_CFC_ (* Continuous Function Chart, elements in execution order *)
#0 INT_TO_REAL(SHU6_P2_TE1_AI1)
#1 DIV(#0, 10)
#2 SHU6_P2_TE1_VN <= #1
#3 I_GT_TE:ISTOK_GT(dost: TRUE, x: #1, ust: SHU6_P2_TE_HIGHLIMIT, shkal: -, gist: 1)
#4 I_LT_TE:ISTOK_LT(dost: TRUE, x: #1, ust: SHU6_P2_TE_LOWLIMIT, shkal: -, gist: 1)
#5 OR(#3.Xb, #4.Xm)
#6 TON_DOST:TON(IN: NOT #5, PT: T#10s)
#7 SHU6_P2_TE1_DOST <= #6.Q
#8 SUB(SHU6_P2_UST_SEZ_LETO, SHU6_P2_UST_SEZ_ZIMA)
#9 fb_SHU6_P2_TE1_B_UST_SEZ_LETO:ISTOK_GT(dost: #6.Q, x: #1, ust: SHU6_P2_UST_SEZ_LETO, shkal: -, gist: #8)
#10 SHU6_P2_TE1_B_UST_SEZ_LETO <= #9.Xb
#11 SHU6_P2_TE1_M_UST_SEZ_LETO <= #9.XbN
#12 fb_SHU6_P2_TE1_B_UST_MYAG_REG:ISTOK_GT(dost: #6.Q, x: #1, ust: SHU6_P2_UST_MYAG_REG, shkal: -, gist: 1)
#13 SHU6_P2_TE1_B_UST_MYAG_REG <= #12.Xb
#14 SHU6_P2_TE1_M_UST_MYAG_REG <= #12.XbN
_END_CFC_
(* the same logic as Structured Text *)
_t75 := INT_TO_REAL(SHU6_P2_TE1_AI1) / 10;
SHU6_P2_TE1_VN := _t75;
I_GT_TE(dost := TRUE, x := _t75, ust := SHU6_P2_TE_HIGHLIMIT, gist := 1);
I_LT_TE(dost := TRUE, x := _t75, ust := SHU6_P2_TE_LOWLIMIT, gist := 1);
TON_DOST(IN := NOT (I_GT_TE.Xb OR I_LT_TE.Xm), PT := T#10s);
SHU6_P2_TE1_DOST := TON_DOST.Q;
fb_SHU6_P2_TE1_B_UST_SEZ_LETO(dost := TON_DOST.Q, x := _t75, ust := SHU6_P2_UST_SEZ_LETO, gist := SHU6_P2_UST_SEZ_LETO - SHU6_P2_UST_SEZ_ZIMA);
SHU6_P2_TE1_B_UST_SEZ_LETO := fb_SHU6_P2_TE1_B_UST_SEZ_LETO.Xb;
SHU6_P2_TE1_M_UST_SEZ_LETO := fb_SHU6_P2_TE1_B_UST_SEZ_LETO.XbN;
fb_SHU6_P2_TE1_B_UST_MYAG_REG(dost := TON_DOST.Q, x := _t75, ust := SHU6_P2_UST_MYAG_REG, gist := 1);
SHU6_P2_TE1_B_UST_MYAG_REG := fb_SHU6_P2_TE1_B_UST_MYAG_REG.Xb;
SHU6_P2_TE1_M_UST_MYAG_REG := fb_SHU6_P2_TE1_B_UST_MYAG_REG.XbN;
END_PROGRAM

(* POU Input/AI/TE4, CFC *)
PROGRAM TE4
VAR
	TE4_YST: REAL;
	fb_TE4: ISTOK_ANALOGVH;
	ofset: REAL;
	fb_SHU6_P2_TE4_M_ZASCH: ISTOK_LT;
	fb_SHU6_P2_TE4_M_UST: ISTOK_LT;
	I_GT_TE: ISTOK_GT;
	I_LT_TE: ISTOK_LT;
	TON_DOST: TON;
END_VAR
VAR (* helpers for the ST form of the networks *)
	_t112 : REAL;
END_VAR
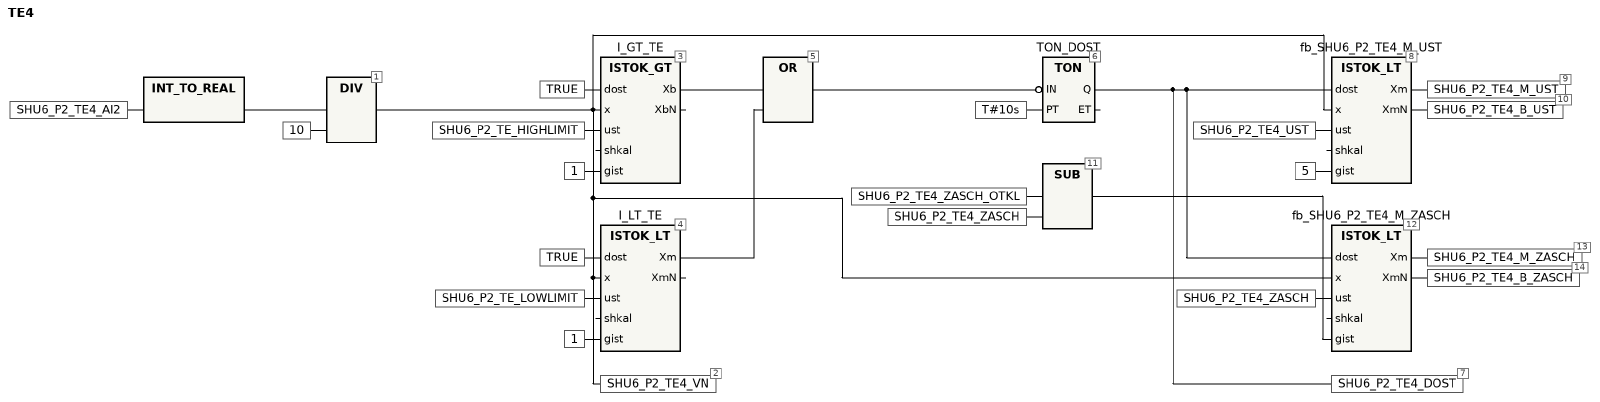
_CFC_ (* Continuous Function Chart, elements in execution order *)
#0 INT_TO_REAL(SHU6_P2_TE4_AI2)
#1 DIV(#0, 10)
#2 SHU6_P2_TE4_VN <= #1
#3 I_GT_TE:ISTOK_GT(dost: TRUE, x: #1, ust: SHU6_P2_TE_HIGHLIMIT, shkal: -, gist: 1)
#4 I_LT_TE:ISTOK_LT(dost: TRUE, x: #1, ust: SHU6_P2_TE_LOWLIMIT, shkal: -, gist: 1)
#5 OR(#3.Xb, #4.Xm)
#6 TON_DOST:TON(IN: NOT #5, PT: T#10s)
#7 SHU6_P2_TE4_DOST <= #6.Q
#8 fb_SHU6_P2_TE4_M_UST:ISTOK_LT(dost: #6.Q, x: #1, ust: SHU6_P2_TE4_UST, shkal: -, gist: 5)
#9 SHU6_P2_TE4_M_UST <= #8.Xm
#10 SHU6_P2_TE4_B_UST <= #8.XmN
#11 SUB(SHU6_P2_TE4_ZASCH_OTKL, SHU6_P2_TE4_ZASCH)
#12 fb_SHU6_P2_TE4_M_ZASCH:ISTOK_LT(dost: #6.Q, x: #1, ust: SHU6_P2_TE4_ZASCH, shkal: -, gist: #11)
#13 SHU6_P2_TE4_M_ZASCH <= #12.Xm
#14 SHU6_P2_TE4_B_ZASCH <= #12.XmN
_END_CFC_
(* the same logic as Structured Text *)
_t112 := INT_TO_REAL(SHU6_P2_TE4_AI2) / 10;
SHU6_P2_TE4_VN := _t112;
I_GT_TE(dost := TRUE, x := _t112, ust := SHU6_P2_TE_HIGHLIMIT, gist := 1);
I_LT_TE(dost := TRUE, x := _t112, ust := SHU6_P2_TE_LOWLIMIT, gist := 1);
TON_DOST(IN := NOT (I_GT_TE.Xb OR I_LT_TE.Xm), PT := T#10s);
SHU6_P2_TE4_DOST := TON_DOST.Q;
fb_SHU6_P2_TE4_M_UST(dost := TON_DOST.Q, x := _t112, ust := SHU6_P2_TE4_UST, gist := 5);
SHU6_P2_TE4_M_UST := fb_SHU6_P2_TE4_M_UST.Xm;
SHU6_P2_TE4_B_UST := fb_SHU6_P2_TE4_M_UST.XmN;
fb_SHU6_P2_TE4_M_ZASCH(dost := TON_DOST.Q, x := _t112, ust := SHU6_P2_TE4_ZASCH, gist := SHU6_P2_TE4_ZASCH_OTKL - SHU6_P2_TE4_ZASCH);
SHU6_P2_TE4_M_ZASCH := fb_SHU6_P2_TE4_M_ZASCH.Xm;
SHU6_P2_TE4_B_ZASCH := fb_SHU6_P2_TE4_M_ZASCH.XmN;
END_PROGRAM

(* POU Input/CI/MV2_1_OB, CFC *)
PROGRAM MV2_1_OB
VAR
	fb_M1_OBRbSM: ISTOK_GT;
	fb_M1b30: ISTOK_GT;
	fb_M1_OBRb45: ISTOK_GT;
	fb_M1_OBRm0_1: ISTOK_LT;
	fb_M_OBR: ISTOK_ANALOGVH;
	ofset: INT := 0;
	SR_DOST_M1: RS;
	dost_ton: TON;
END_VAR
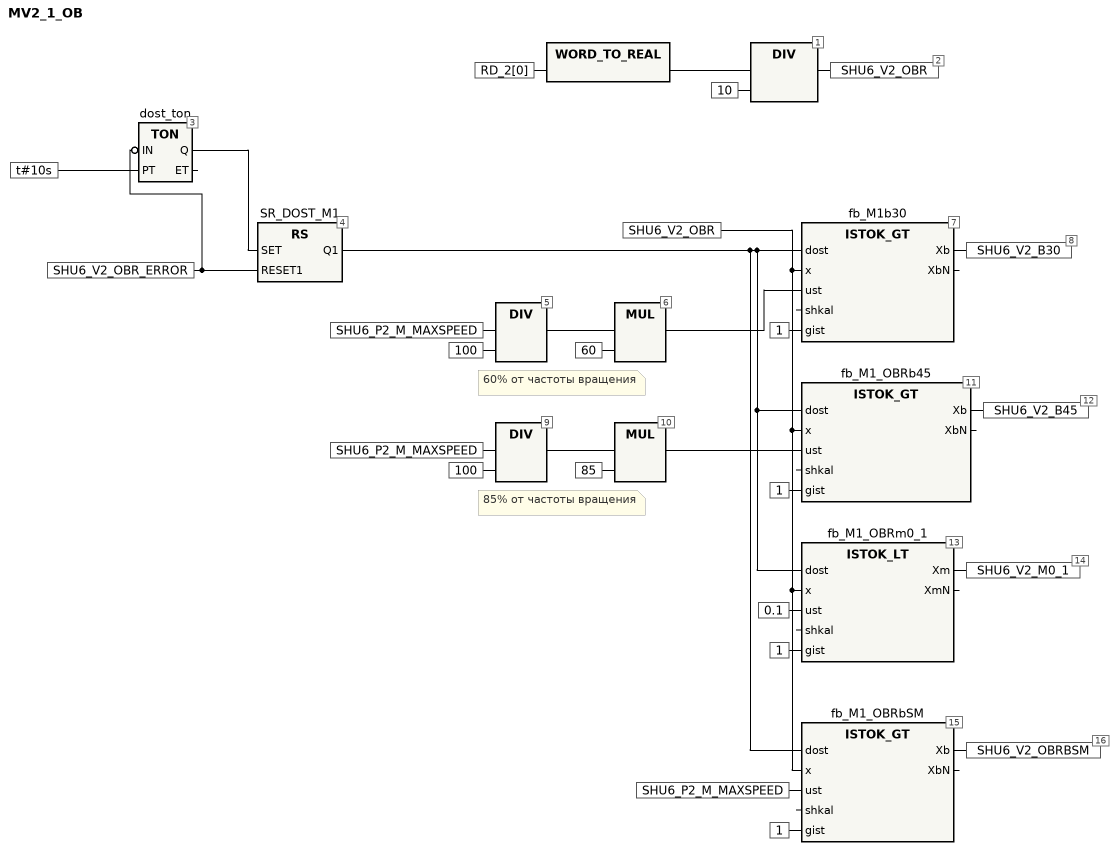
_CFC_ (* Continuous Function Chart, elements in execution order *)
(* 85% от частоты вращения *)
(* 60% от частоты вращения *)
#0 WORD_TO_REAL(RD_2[0])
#1 DIV(#0, 10)
#2 SHU6_V2_OBR <= #1
#3 dost_ton:TON(IN: NOT SHU6_V2_OBR_ERROR, PT: t#10s)
#4 SR_DOST_M1:RS(SET: #3.Q, RESET1: SHU6_V2_OBR_ERROR)
#5 DIV(SHU6_P2_M_MAXSPEED, 100)
#6 MUL(#5, 60)
#7 fb_M1b30:ISTOK_GT(dost: #4.Q1, x: SHU6_V2_OBR, ust: #6, shkal: -, gist: 1)
#8 SHU6_V2_B30 <= #7.Xb
#9 DIV(SHU6_P2_M_MAXSPEED, 100)
#10 MUL(#9, 85)
#11 fb_M1_OBRb45:ISTOK_GT(dost: #4.Q1, x: SHU6_V2_OBR, ust: #10, shkal: -, gist: 1)
#12 SHU6_V2_B45 <= #11.Xb
#13 fb_M1_OBRm0_1:ISTOK_LT(dost: #4.Q1, x: SHU6_V2_OBR, ust: 0.1, shkal: -, gist: 1)
#14 SHU6_V2_M0_1 <= #13.Xm
#15 fb_M1_OBRbSM:ISTOK_GT(dost: #4.Q1, x: SHU6_V2_OBR, ust: SHU6_P2_M_MAXSPEED, shkal: -, gist: 1)
#16 SHU6_V2_OBRBSM <= #15.Xb
_END_CFC_
(* the same logic as Structured Text *)
(* 85% от частоты вращения *)
(* 60% от частоты вращения *)
SHU6_V2_OBR := WORD_TO_REAL(RD_2[0]) / 10;
dost_ton(IN := NOT SHU6_V2_OBR_ERROR, PT := t#10s);
SR_DOST_M1(SET := dost_ton.Q, RESET1 := SHU6_V2_OBR_ERROR);
fb_M1b30(dost := SR_DOST_M1.Q1, x := SHU6_V2_OBR, ust := (SHU6_P2_M_MAXSPEED / 100) * 60, gist := 1);
SHU6_V2_B30 := fb_M1b30.Xb;
fb_M1_OBRb45(dost := SR_DOST_M1.Q1, x := SHU6_V2_OBR, ust := (SHU6_P2_M_MAXSPEED / 100) * 85, gist := 1);
SHU6_V2_B45 := fb_M1_OBRb45.Xb;
fb_M1_OBRm0_1(dost := SR_DOST_M1.Q1, x := SHU6_V2_OBR, ust := 0.1, gist := 1);
SHU6_V2_M0_1 := fb_M1_OBRm0_1.Xm;
fb_M1_OBRbSM(dost := SR_DOST_M1.Q1, x := SHU6_V2_OBR, ust := SHU6_P2_M_MAXSPEED, gist := 1);
SHU6_V2_OBRBSM := fb_M1_OBRbSM.Xb;
END_PROGRAM

(* POU Input/AI/TE6_T, CFC *)
PROGRAM TE6_T
VAR
	fb_UE3_T: ISTOK_ANALOGVH;
	ofset: REAL;
	fb_SHU6_P2_TE6_T_NEQ_UST: ISTOK_EQ;
	fb_TE6_m_UST: ISTOK_LT;
	fb_TE6_b_UST: ISTOK_GT;
	I_GT_TE6: ISTOK_GT;
	I_LT_TE6: ISTOK_LT;
	TON_DOST: TON;
END_VAR
VAR (* helpers for the ST form of the networks *)
	_t108 : REAL;
END_VAR
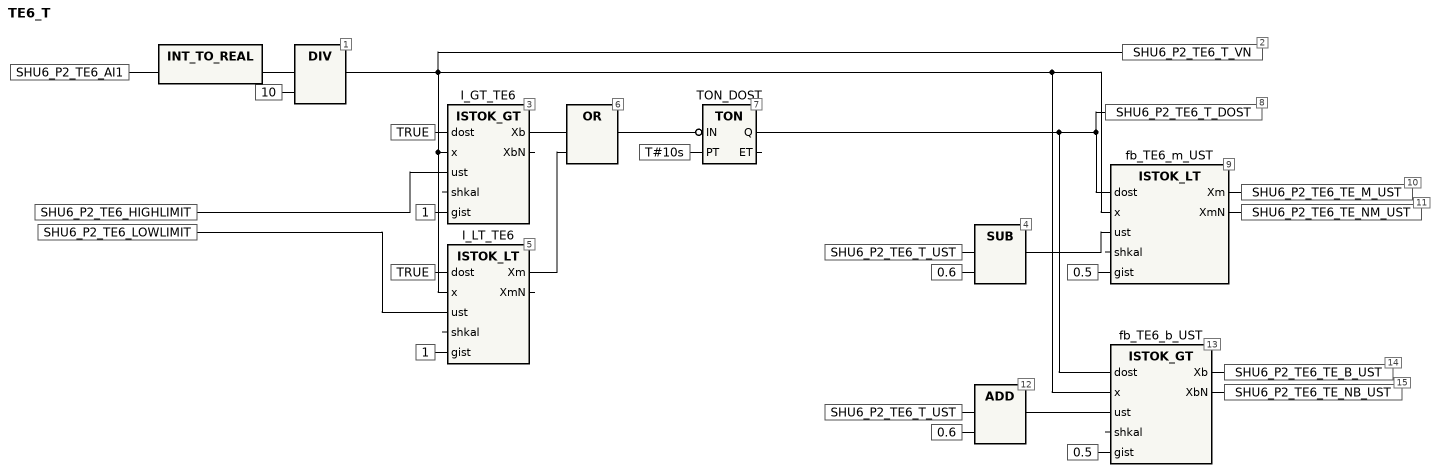
